FUNCTION_BLOCK IntToBin (* Basic Function Block Type *)
  (* Standard: 61499-2 *)
  (* Version 0.0, 21/06/2022, Lernfabrik, WBK hackaton, Template *)
  PACKAGE Main;
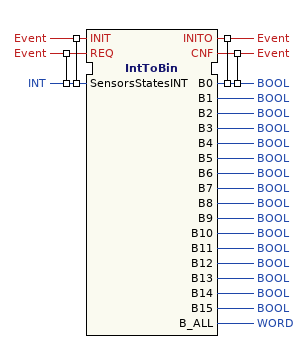
  EVENT_INPUT
    INIT WITH SensorsStatesINT; (* Initialization Request *)
    REQ WITH SensorsStatesINT; (* Normal Execution Request *)
  END_EVENT
  EVENT_OUTPUT
    INITO WITH B0; (* Initialization Confirm *)
    CNF WITH B0; (* Execution Confirmation *)
  END_EVENT
  VAR_INPUT
    SensorsStatesINT : INT; (* Input event qualifier *)
  END_VAR
  VAR_OUTPUT
    B0 : BOOL; (* Output event qualifier *)
    B1 : BOOL;
    B2 : BOOL;
    B3 : BOOL;
    B4 : BOOL;
    B5 : BOOL;
    B6 : BOOL;
    B7 : BOOL;
    B8 : BOOL;
    B9 : BOOL;
    B10 : BOOL;
    B11 : BOOL;
    B12 : BOOL;
    B13 : BOOL;
    B14 : BOOL;
    B15 : BOOL;
    B_ALL : WORD;
  END_VAR
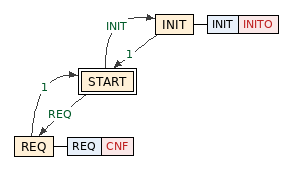
  EC_STATES
    START; (* Initial State *)
    INIT : INIT -> INITO; (* Initialization *)
    REQ : REQ -> CNF; (* Normal execution *)
  END_STATES
  EC_TRANSITIONS
    START TO INIT := INIT;
    INIT TO START := 1;
    START TO REQ := REQ;
    REQ TO START := 1;
  END_TRANSITIONS
  ALGORITHM INIT IN ST: (* Initialization algorithm *)
;
  END_ALGORITHM
  ALGORITHM REQ IN ST: (* Normally executed algorithm *)
;
  END_ALGORITHM
END_FUNCTION_BLOCK
